TYPE "Analogic_SensorManagement_Data"
VERSION : 0.1
// Block: Analogic_SensorManagement_Data
   STRUCT
      OffsetValue : LReal;
      OffsetValid : Bool;
   END_STRUCT;

END_TYPE
